PROGRAM MAIN
VAR
	
END_VAR

END_PROGRAM

(* stored: Version 1.1.0.1, ProductVersion 3.1.4024.16
   POU MAIN: Id {a80238dd-9798-4b30-974d-cc9fee391c36}, SpecialFunc None *)
